FUNCTION_BLOCK FB_Interface_MbRtu
VAR_INPUT
	UnitID			: BYTE;
	bExecute		: BOOL;
	bStop			: BOOL;
	bReset			: BOOL;
	idDevice		: UINT;
	fTargetSpeed	: REAL;
END_VAR
VAR_OUTPUT
END_VAR
VAR
	tmp				: WORD;
	bFB_Stop		: BOOL;
	Address1		: WORD;
	Address2		: WORD;
	Address3		: WORD;
	WriteVal  		: WORD;
	WriteVal2		: ARRAY [1..2] OF WORD;
	nState			: INT;
	fbTimer			: TON;
	nStateAll		: INT;
END_VAR

CASE nStateAll OF
	0:
		t := 1;
		nStateAll := 1;
	1:
		IF UnitID = t THEN
			IF idDevice = 1 THEN
				IF WriteVal <> REAL_TO_WORD(fTargetSpeed*100) THEN
					WriteVal := REAL_TO_WORD(fTargetSpeed*100);
					nStateAll := 2;
				ELSE 
					nStateAll := 9;
				END_IF
			ELSIF idDevice = 2 THEN
				IF WriteVal2[1] <> REAL_TO_WORD(fTargetSpeed) THEN
					WriteVal2[1] := REAL_TO_WORD(fTargetSpeed);
					nStateAll := 3;
				ELSE
					nStateAll := 9;
				END_IF
			END_IF
		END_IF
	2:
		fbTimer(IN := TRUE, PT := T#100MS);
		fbModbus.WriteRegs(
						UnitID:= UnitID, 
						Quantity:= 1, 
						MBAddr:= 8193, 
						cbLength:= SIZEOF(WriteVal), 
						pMemoryAddr:=  ADR(WriteVal), 
						Execute:= TRUE, 
						Timeout:= T#1S, 
						BUSY=> Busy[UnitID], 
						Error=> Error[UnitID], 
						ErrorId=> ErrorID[UnitID] , 
						cbRead=> );
		IF fbTimer.Q AND NOT Busy[UnitID] THEN
			nStateAll := 9;
		END_IF
	3:
		fbTimer(IN := TRUE, PT := T#100MS);
		fbModbus.WriteRegs(
						UnitID:= UnitID, 
						Quantity:= 2, 
						MBAddr:= 1034, 
						cbLength:= SIZEOF(WriteVal2), 
						pMemoryAddr:=  ADR(WriteVal2), 
						Execute:= TRUE, 
						Timeout:= T#1S, 
						BUSY=> Busy[UnitID], 
						Error=> Error[UnitID], 
						ErrorId=> ErrorID[UnitID], 
						cbRead=> );
		IF fbTimer.Q AND NOT Busy[UnitID] THEN
			nStateAll := 9;	
		END_IF			
	9:
		fbTimer(IN := false);
		fbModbus.WriteRegs(Execute := FALSE);
		t := t + 1;
		nStateAll := 11;
	11:
		IF t > 7 THEN
			t := 1;
			nStateAll := 1;
		ELSE
			nStateAll := 1;
		END_IF	
END_CASE

END_FUNCTION_BLOCK

(* stored: Version 1.1.0.1, ProductVersion 3.1.4024.12
   POU FB_Interface_MbRtu: Id {b83d9a67-33c8-4e92-84f1-2ed0fa6af340}, SpecialFunc None *)
